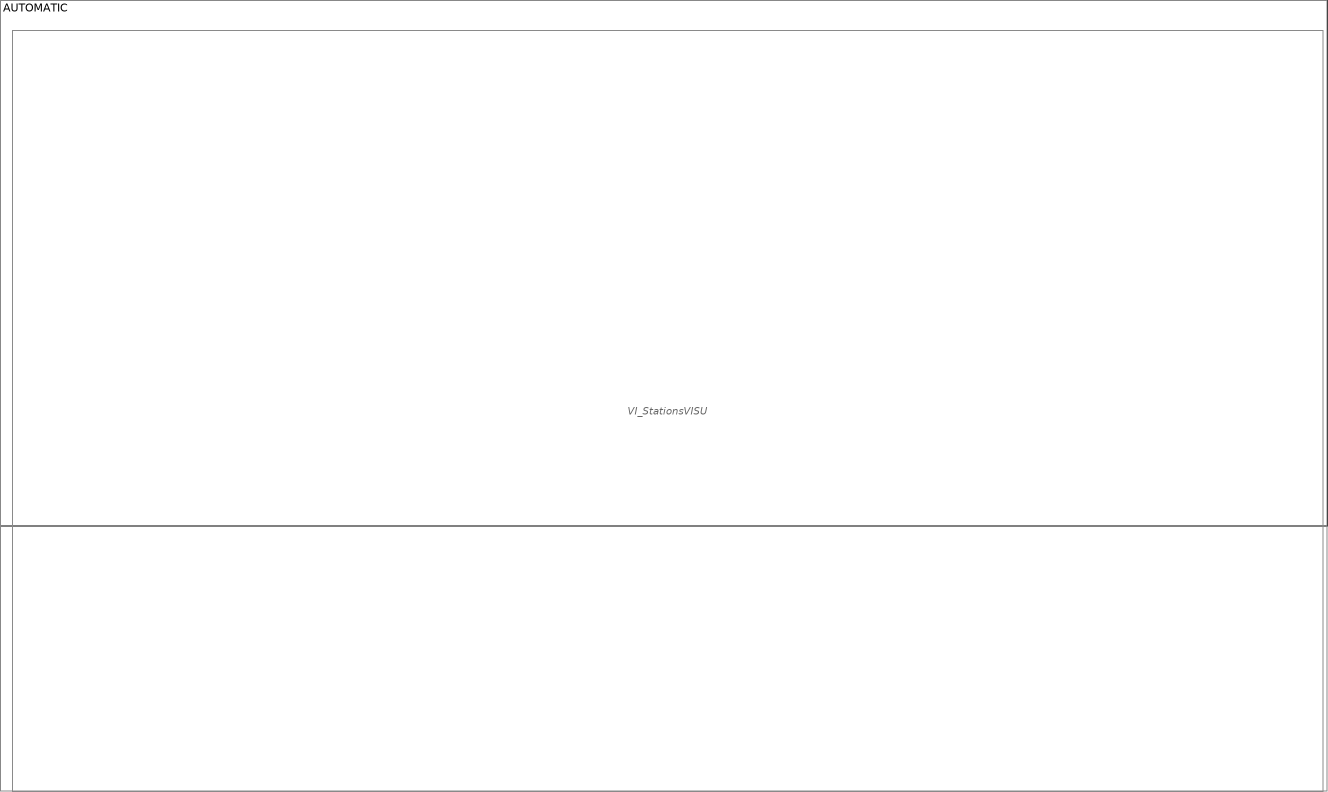
VISUALIZATION VI_XTSAutoVisu  // 1328x792
VAR_IN_OUT
	xts : XTS_System;
END_VAR
VAR
	stTableStruct : ARRAY [1..25] OF stTableStructx10;
END_VAR
    Rectangle (0,0 1328x526), "AUTOMATIC"
    Frame (12,30 1311x762)
        shows VI_StationsVISU(aStations := xts.aStations)
END_VISUALIZATION

(* stored: Version 1.1.0.1, ProductVersion 3.1.4024.11
   Visu VI_XTSAutoVisu: Id {f9e20e03-8613-4e3e-8212-6b9c477a923d} *)
